{attribute 'qualified_only'}
{attribute 'strict'}
TYPE enum_DriveUpdateError :
(
	NoError,
	FileNotFound,
	FileClosedFailed,
	FoeFailed
);
END_TYPE

(* stored: Version 1.1.0.1, ProductVersion 3.1.4024.3
   DUT enum_DriveUpdateError: Id {896e3fea-e556-0bfc-34c9-6642dbbf2232} *)
